FUNCTION CEIL (* This is a rounding function which returns the smallest possible integer which is greater or equal to X. *)
  (* Standard: 61499-1 *)
  (* Version 1.0, 2026-09-17, Franz Höpfinger, Portiert aus OSCAT_basic CEIL.TcPOU - Bereichspruefung (X >= 32767.0 / X <= -32768.0) schuetzt vor INT-Ueberlauf. *)
  PACKAGE OSCAT::Basic::POUs::Mathematical;
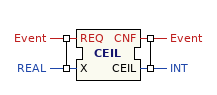
  EVENT_INPUT
    REQ WITH X;
  END_EVENT
  EVENT_OUTPUT
    CNF WITH CEIL;
  END_EVENT
  VAR_INPUT
    X : REAL;
  END_VAR
  VAR_OUTPUT
    CEIL : INT;
  END_VAR
  BODY IN ST:
PACKAGE OSCAT::Basic::POUs::Mathematical;

(* This is a rounding function which returns the smallest possible integer which is greater or equal to X (clamped to INT range -32768..32767). *)
FUNCTION CEIL : INT
VAR_INPUT
	X : REAL;
END_VAR

(*
 * version 1.1	21. mar. 2008 programmer 	hugo tested by		tobias
 * *
 * This is a rounding function which returns the smallest possible integer which is greater or equal to X.
 * ceil(3.14) = 4 ceil(-3.14) = -3
 * Portiert 2026-09-17: Bereichspruefung schuetzt vor INT-Ueberlauf.
 *)
IF X >= 32767.0 THEN
	CEIL := 32767;
ELSIF X <= -32768.0 THEN
	CEIL := -32768;
ELSE
	CEIL := REAL_TO_INT(X);
	IF CEIL < X THEN
		CEIL := CEIL + 1;
	END_IF;
END_IF;

END_FUNCTION

(* revision history hm	7. feb. 2007	rev 1.0 original version
 * *
 * hm	21. mar. 2008	rev 1.1 use REAL_TO_INT instead of trunc for compatibility reasons *)
  END_BODY
END_FUNCTION
